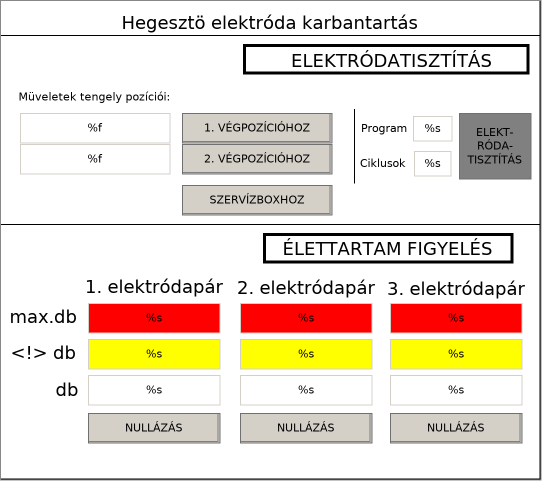
VISUALIZATION Hegesztes_Karbantartas  // 542x481
    Rectangle (0,-1 540x480)
    Textfield (20,113 150x30), "%f", text variable: GVL.lrCsiszoloPosition1
        OnMouseClick: write the text variable via VisuDialogs.Numpad, min -10000, max -1
    Button (182,113 150x30), "1. VÉGPOZÍCIÓHOZ"
        OnMouseUp: execute { JOZSITENGELY.lrJozsiPosition:=GVL.lrCsiszoloPosition1; JOZSITENGELY.sJozsiAxisCommand:='MOVE'; }
    Textfield (20,144 150x30), "%f", text variable: GVL.lrCsiszoloPosition2
        OnMouseClick: write the text variable via VisuDialogs.Numpad, min -10000, max -1
    Button (182,144 150x30), "2. VÉGPOZÍCIÓHOZ"
        OnMouseUp: execute { JOZSITENGELY.lrJozsiPosition:=GVL.lrCsiszoloPosition2; JOZSITENGELY.sJozsiAxisCommand:='MOVE'; }
    Textfield (88,303 132x30), "%s", text variable: GVL.nElectrode1UsageMax
        OnMouseClick: write the text variable via VisuDialogs.Numpad, min 1, max 100000
    Button (88,413 132x30), "NULLÁZÁS"
        OnMouseUp: execute { GVL.nElectrode1Usage:=0; }
    Button (182,185 150x30), "SZERVÍZBOXHOZ"
        OnMouseUp: execute { JOZSITENGELY.lrJozsiPosition:=GVL.lrNTCSzervizbox; JOZSITENGELY.sJozsiAxisCommand:='MOVE'; }
    Button (459,113 72x66), "ELEKT- RÓDA- TISZTÍTÁS"
        OnMouseUp: execute {
            IF GVL.bJOZSITENGELYReserved=FALSE THEN
            	HEGESZTOFEJTISZTITAS.iState:=1;
            END_IF;
        }
    Line (0,35) (540,35), "Hegesztö elektróda karbantartás"
    Line (0,224) (540,224)
    RoundedRectangle (263,233 250x30)
    Label (255,234 265x30), "ÉLETTARTAM FIGYELÉS"
    Label (13,82 163x30), "Müveletek tengely pozíciói:"
    Textfield (413,116 39x25), "%s", text variable: GVL.nHegFejTisztProgram
        OnMouseClick: write the text variable via VisuDialogs.Numpad, min 11, max 14
    Textfield (414,151 37x25), "%s", text variable: GVL.nHegFejTisztCiklusok
        OnMouseClick: write the text variable via VisuDialogs.Numpad, min 1, max 20
    Label (358,116 54x25), "Program"
    Label (357,151 54x25), "Ciklusok"
    Line (354,109) (354,183)
    RoundedRectangle (243,44 286x30)
    Label (255,46 273x30), "ELEKTRÓDATISZTÍTÁS"
    Label (81,272 146x30), "1. elektródapár"
    Label (233,273 146x30), "2. elektródapár"
    Label (383,274 146x30), "3. elektródapár"
    Textfield (88,375 132x30), "%s", text variable: GVL.nElectrode1Usage, colour toggle: GVL.nElectrode1Usage>GVL.nElectrode1UsageWarn
        p2167032090: GVL.nElectrode1AlarmColor
    Textfield (240,303 132x30), "%s", text variable: GVL.nElectrode2UsageMax
        OnMouseClick: write the text variable via VisuDialogs.Numpad, min 1, max 100000
    Button (240,413 132x30), "NULLÁZÁS"
        OnMouseUp: execute { GVL.nElectrode2Usage:=0; }
    Textfield (240,375 132x30), "%s", text variable: GVL.nElectrode2Usage, colour toggle: GVL.nElectrode2Usage>GVL.nElectrode2UsageWarn
        p2167032090: GVL.nElectrode2AlarmColor
    Textfield (390,303 132x30), "%s", text variable: GVL.nElectrode3UsageMax
        OnMouseClick: write the text variable via VisuDialogs.Numpad, min 1, max 100000
    Button (390,413 132x30), "NULLÁZÁS"
        OnMouseUp: execute { GVL.nElectrode3Usage:=0; }
    Textfield (390,375 132x30), "%s", text variable: GVL.nElectrode3Usage, colour toggle: GVL.nElectrode3Usage>GVL.nElectrode3UsageWarn
        p2167032090: GVL.nElectrode3AlarmColor
    Label (5,302 77x30), "max.db"
    Label (52,375 30x30), "db"
    Label (5,338 77x30), "<!> db"
    Textfield (88,339 132x30), "%s", text variable: GVL.nElectrode1UsageWarn
        OnMouseClick: write the text variable via VisuDialogs.Numpad, min 1, max 100000
    Textfield (240,339 132x30), "%s", text variable: GVL.nElectrode2UsageWarn
        OnMouseClick: write the text variable via VisuDialogs.Numpad, min 1, max 100000
    Textfield (390,339 132x30), "%s", text variable: GVL.nElectrode3UsageWarn
        OnMouseClick: write the text variable via VisuDialogs.Numpad, min 1, max 100000
END_VISUALIZATION

(* stored: Version 1.1.0.1, ProductVersion 3.1.4024.11
   Visu Hegesztes_Karbantartas: Id {605d404f-037f-421a-98a0-199ebd543b95} *)
